Fanuc TP program (LS listing): DISTI_LINE_V1.LS

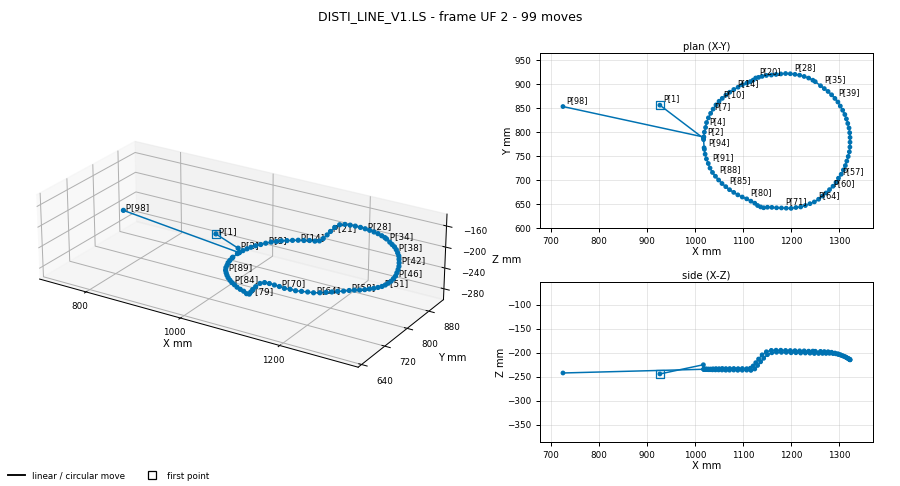
[picture p0: tool path of DISTI_LINE_V1.LS in frame UF 2, 99 of 99 moves have a stored position in this frame; points joined in program order, loops and branches not executed]
/PROG  DISTI_LINE_V1
/ATTR
OWNER		= MNEDITOR;
COMMENT		= "WeldPRO Auto-Gen";
PROG_SIZE	= 7109;
CREATE		= DATE 26-07-21  TIME 17:58:54;
MODIFIED	= DATE 26-07-21  TIME 18:14:06;
FILE_NAME	= DISTI_LI;
VERSION		= 0;
LINE_COUNT	= 113;
MEMORY_SIZE	= 7429;
PROTECT		= READ_WRITE;
TCD:  STACK_SIZE	= 0,
      TASK_PRIORITY	= 50,
      TIME_SLICE	= 0,
      BUSY_LAMP_OFF	= 0,
      ABORT_REQUEST	= 0,
      PAUSE_REQUEST	= 0;
DEFAULT_GROUP	= 1,*,*,*,*;
CONTROL_CODE	= 00000000 00000000;
/APPL
/MN
   1:  !WeldPRO Auto-Generated TPP ;
   2:  !Tor XL_176 _2, Feature1 ;
   3:   ;
   4:  UFRAME_NUM=2 ;
   5:  UTOOL_NUM=2 ;
   6:L P[1] 100mm/sec FINE    ;
   7:   ;
   8:  !Segment1 ;
   9:L P[2] 100mm/sec FINE    ;
  10:  CALL LASER_OFF    ;
  11:   ;
  12:L P[99] R[23:moving]mm/sec CNT100    ;
  13:   ;
  14:L P[3] R[23:moving]mm/sec CNT100    ;
  15:L P[4] R[23:moving]mm/sec CNT100    ;
  16:L P[5] R[23:moving]mm/sec CNT100    ;
  17:L P[6] R[23:moving]mm/sec CNT100    ;
  18:L P[7] R[23:moving]mm/sec CNT100    ;
  19:L P[8] R[23:moving]mm/sec CNT100    ;
  20:L P[9] R[23:moving]mm/sec CNT100    ;
  21:L P[10] R[23:moving]mm/sec CNT100    ;
  22:L P[11] R[23:moving]mm/sec CNT100    ;
  23:L P[12] R[23:moving]mm/sec CNT100    ;
  24:L P[13] R[23:moving]mm/sec CNT100    ;
  25:L P[14] R[23:moving]mm/sec CNT100    ;
  26:L P[15] R[23:moving]mm/sec CNT100    ;
  27:L P[16] R[23:moving]mm/sec CNT100    ;
  28:L P[17] R[23:moving]mm/sec CNT100    ;
  29:L P[18] R[23:moving]mm/sec CNT100    ;
  30:L P[19] R[23:moving]mm/sec CNT100    ;
  31:L P[20] R[23:moving]mm/sec CNT100    ;
  32:L P[21] R[23:moving]mm/sec CNT100    ;
  33:L P[22] R[23:moving]mm/sec CNT100    ;
  34:L P[23] R[23:moving]mm/sec CNT100    ;
  35:L P[24] R[23:moving]mm/sec CNT100    ;
  36:L P[25] R[23:moving]mm/sec CNT100    ;
  37:L P[26] R[23:moving]mm/sec CNT100    ;
  38:L P[27] R[23:moving]mm/sec CNT100    ;
  39:L P[28] R[23:moving]mm/sec CNT100    ;
  40:L P[29] R[23:moving]mm/sec CNT100    ;
  41:L P[30] R[23:moving]mm/sec CNT100    ;
  42:L P[31] R[23:moving]mm/sec CNT100    ;
  43:L P[32] R[23:moving]mm/sec CNT100    ;
  44:L P[33] R[23:moving]mm/sec CNT100    ;
  45:L P[34] R[23:moving]mm/sec CNT100    ;
  46:L P[35] R[23:moving]mm/sec CNT100    ;
  47:L P[36] R[23:moving]mm/sec CNT100    ;
  48:L P[37] R[23:moving]mm/sec CNT100    ;
  49:L P[38] R[23:moving]mm/sec CNT100    ;
  50:L P[39] R[23:moving]mm/sec CNT100    ;
  51:L P[40] R[23:moving]mm/sec CNT100    ;
  52:L P[41] R[23:moving]mm/sec CNT100    ;
  53:L P[42] R[23:moving]mm/sec CNT100    ;
  54:L P[43] R[23:moving]mm/sec CNT100    ;
  55:L P[44] R[23:moving]mm/sec CNT100    ;
  56:L P[45] R[23:moving]mm/sec CNT100    ;
  57:L P[46] R[23:moving]mm/sec CNT100    ;
  58:L P[47] R[23:moving]mm/sec CNT100    ;
  59:L P[48] R[23:moving]mm/sec CNT100    ;
  60:L P[49] R[23:moving]mm/sec CNT100    ;
  61:L P[50] R[23:moving]mm/sec CNT100    ;
  62:L P[51] R[23:moving]mm/sec CNT100    ;
  63:L P[52] R[23:moving]mm/sec CNT100    ;
  64:L P[53] R[23:moving]mm/sec CNT100    ;
  65:L P[54] R[23:moving]mm/sec CNT100    ;
  66:L P[55] R[23:moving]mm/sec CNT100    ;
  67:L P[56] R[23:moving]mm/sec CNT100    ;
  68:L P[57] R[23:moving]mm/sec CNT100    ;
  69:L P[58] R[23:moving]mm/sec CNT100    ;
  70:L P[59] R[23:moving]mm/sec CNT100    ;
  71:L P[60] R[23:moving]mm/sec CNT100    ;
  72:L P[61] R[23:moving]mm/sec CNT100    ;
  73:L P[62] R[23:moving]mm/sec CNT100    ;
  74:L P[63] R[23:moving]mm/sec CNT100    ;
  75:L P[64] R[23:moving]mm/sec CNT100    ;
  76:L P[65] R[23:moving]mm/sec CNT100    ;
  77:L P[66] R[23:moving]mm/sec CNT100    ;
  78:L P[67] R[23:moving]mm/sec CNT100    ;
  79:L P[68] R[23:moving]mm/sec CNT100    ;
  80:L P[69] R[23:moving]mm/sec CNT100    ;
  81:L P[70] R[23:moving]mm/sec CNT100    ;
  82:L P[71] R[23:moving]mm/sec CNT100    ;
  83:L P[72] R[23:moving]mm/sec CNT100    ;
  84:L P[73] R[23:moving]mm/sec CNT100    ;
  85:L P[74] R[23:moving]mm/sec CNT100    ;
  86:L P[75] R[23:moving]mm/sec CNT100    ;
  87:L P[76] R[23:moving]mm/sec CNT100    ;
  88:L P[77] R[23:moving]mm/sec CNT100    ;
  89:L P[78] R[23:moving]mm/sec CNT100    ;
  90:L P[79] R[23:moving]mm/sec CNT100    ;
  91:L P[80] R[23:moving]mm/sec CNT100    ;
  92:L P[81] R[23:moving]mm/sec CNT100    ;
  93:L P[82] R[23:moving]mm/sec CNT100    ;
  94:L P[83] R[23:moving]mm/sec CNT100    ;
  95:L P[84] R[23:moving]mm/sec CNT100    ;
  96:L P[85] R[23:moving]mm/sec CNT100    ;
  97:L P[86] R[23:moving]mm/sec CNT100    ;
  98:L P[87] R[23:moving]mm/sec CNT100    ;
  99:L P[88] R[23:moving]mm/sec CNT100    ;
 100:L P[89] R[23:moving]mm/sec CNT100    ;
 101:L P[90] R[23:moving]mm/sec CNT100    ;
 102:L P[91] R[23:moving]mm/sec CNT100    ;
 103:L P[92] R[23:moving]mm/sec CNT100    ;
 104:L P[93] R[23:moving]mm/sec CNT100    ;
 105:L P[94] R[23:moving]mm/sec CNT100    ;
 106:L P[95] R[23:moving]mm/sec CNT100    ;
 107:L P[96] R[23:moving]mm/sec CNT100    ;
 108:L P[97] R[23:moving]mm/sec FINE    ;
 109:  CALL LASER_OFF    ;
 110:   ;
 111:  !Feature Retreat ;
 112:L P[98] 100mm/sec FINE    ;
 113:  CALL ROTATE    ;
/POS
P[1]{
   GP1:
	UF : 2, UT : 2,		CONFIG : 'F D T, 0, 0, 0',
	X =   927.346  mm,	Y =   856.354  mm,	Z =  -244.034  mm,
	W =  -106.482 deg,	P =   -15.198 deg,	R =    86.345 deg
};
P[2]{
   GP1:
	UF : 2, UT : 2,		CONFIG : 'F D T, 0, 0, 0',
	X =  1017.849  mm,	Y =   787.602  mm,	Z =  -224.873  mm,
	W =  -106.491 deg,	P =   -15.193 deg,	R =    86.327 deg
};
P[3]{
   GP1:
	UF : 2, UT : 2,		CONFIG : 'F D T, 0, 0, 0',
	X =  1019.935  mm,	Y =   800.294  mm,	Z =  -233.990  mm,
	W =  -106.460 deg,	P =   -15.318 deg,	R =    81.648 deg
};
P[4]{
   GP1:
	UF : 2, UT : 2,		CONFIG : 'F D T, 0, 0, 0',
	X =  1022.444  mm,	Y =   809.956  mm,	Z =  -233.523  mm,
	W =  -106.425 deg,	P =   -15.445 deg,	R =    76.281 deg
};
P[5]{
   GP1:
	UF : 2, UT : 2,		CONFIG : 'F D T, 0, 0, 0',
	X =  1024.421  mm,	Y =   820.142  mm,	Z =  -233.847  mm,
	W =  -106.381 deg,	P =   -15.559 deg,	R =    71.464 deg
};
P[6]{
   GP1:
	UF : 2, UT : 2,		CONFIG : 'F D T, 0, 0, 0',
	X =  1028.297  mm,	Y =   829.982  mm,	Z =  -233.703  mm,
	W =  -106.310 deg,	P =   -15.698 deg,	R =    65.272 deg
};
P[7]{
   GP1:
	UF : 2, UT : 2,		CONFIG : 'F D T, 0, 0, 0',
	X =  1032.934  mm,	Y =   839.356  mm,	Z =  -233.745  mm,
	W =  -106.251 deg,	P =   -15.795 deg,	R =    60.811 deg
};
P[8]{
   GP1:
	UF : 2, UT : 2,		CONFIG : 'F D T, 0, 0, 0',
	X =  1038.061  mm,	Y =   848.132  mm,	Z =  -233.295  mm,
	W =  -106.174 deg,	P =   -15.897 deg,	R =    55.794 deg
};
P[9]{
   GP1:
	UF : 2, UT : 2,		CONFIG : 'F D T, 0, 0, 0',
	X =  1044.053  mm,	Y =   856.873  mm,	Z =  -232.984  mm,
	W =  -106.090 deg,	P =   -15.988 deg,	R =    50.970 deg
};
P[10]{
   GP1:
	UF : 2, UT : 2,		CONFIG : 'F D T, 0, 0, 0',
	X =  1050.502  mm,	Y =   864.509  mm,	Z =  -233.095  mm,
	W =  -106.027 deg,	P =   -16.056 deg,	R =    47.314 deg
};
P[11]{
   GP1:
	UF : 2, UT : 2,		CONFIG : 'F D T, 0, 0, 0',
	X =  1057.143  mm,	Y =   870.540  mm,	Z =  -232.650  mm,
	W =  -105.939 deg,	P =   -16.126 deg,	R =    42.935 deg
};
P[12]{
   GP1:
	UF : 2, UT : 2,		CONFIG : 'F D T, 0, 0, 0',
	X =  1064.674  mm,	Y =   877.253  mm,	Z =  -232.934  mm,
	W =  -105.872 deg,	P =   -16.175 deg,	R =    39.733 deg
};
P[13]{
   GP1:
	UF : 2, UT : 2,		CONFIG : 'F D T, 0, 0, 0',
	X =  1072.654  mm,	Y =   883.324  mm,	Z =  -232.851  mm,
	W =  -105.783 deg,	P =   -16.243 deg,	R =    35.484 deg
};
P[14]{
   GP1:
	UF : 2, UT : 2,		CONFIG : 'F D T, 0, 0, 0',
	X =  1081.152  mm,	Y =   888.974  mm,	Z =  -232.722  mm,
	W =  -105.683 deg,	P =   -16.290 deg,	R =    31.072 deg
};
P[15]{
   GP1:
	UF : 2, UT : 2,		CONFIG : 'F D T, 0, 0, 0',
	X =  1090.115  mm,	Y =   893.784  mm,	Z =  -232.991  mm,
	W =  -105.584 deg,	P =   -16.329 deg,	R =    26.914 deg
};
P[16]{
   GP1:
	UF : 2, UT : 2,		CONFIG : 'F D T, 0, 0, 0',
	X =  1098.940  mm,	Y =   898.687  mm,	Z =  -232.748  mm,
	W =  -105.545 deg,	P =   -16.341 deg,	R =    25.103 deg
};
P[17]{
   GP1:
	UF : 2, UT : 2,		CONFIG : 'F D T, 0, 0, 0',
	X =  1107.970  mm,	Y =   902.159  mm,	Z =  -233.094  mm,
	W =  -115.468 deg,	P =   -16.090 deg,	R =    30.046 deg
};
P[18]{
   GP1:
	UF : 2, UT : 2,		CONFIG : 'F D T, 0, 0, 0',
	X =  1115.546  mm,	Y =   905.308  mm,	Z =  -232.090  mm,
	W =  -126.721 deg,	P =   -15.366 deg,	R =    26.538 deg
};
P[19]{
   GP1:
	UF : 2, UT : 2,		CONFIG : 'F D T, 0, 0, 0',
	X =  1121.367  mm,	Y =   908.505  mm,	Z =  -227.368  mm,
	W =  -119.393 deg,	P =   -15.981 deg,	R =    16.221 deg
};
P[20]{
   GP1:
	UF : 2, UT : 2,		CONFIG : 'F D T, 0, 0, 0',
	X =  1126.751  mm,	Y =   912.917  mm,	Z =  -220.637  mm,
	W =  -115.329 deg,	P =   -16.208 deg,	R =    11.788 deg
};
P[21]{
   GP1:
	UF : 2, UT : 2,		CONFIG : 'F D T, 0, 0, 0',
	X =  1132.715  mm,	Y =   914.254  mm,	Z =  -213.028  mm,
	W =  -112.690 deg,	P =   -16.313 deg,	R =     9.687 deg
};
P[22]{
   GP1:
	UF : 2, UT : 2,		CONFIG : 'F D T, 0, 0, 0',
	X =  1140.073  mm,	Y =   916.305  mm,	Z =  -204.283  mm,
	W =  -110.089 deg,	P =   -16.384 deg,	R =     9.676 deg
};
P[23]{
   GP1:
	UF : 2, UT : 2,		CONFIG : 'F D T, 0, 0, 0',
	X =  1148.969  mm,	Y =   918.238  mm,	Z =  -197.811  mm,
	W =  -107.448 deg,	P =   -16.428 deg,	R =     8.430 deg
};
P[24]{
   GP1:
	UF : 2, UT : 2,		CONFIG : 'F D T, 0, 0, 0',
	X =  1159.237  mm,	Y =   919.017  mm,	Z =  -194.999  mm,
	W =  -105.451 deg,	P =   -16.442 deg,	R =     6.850 deg
};
P[25]{
   GP1:
	UF : 2, UT : 2,		CONFIG : 'F D T, 0, 0, 0',
	X =  1169.084  mm,	Y =   920.317  mm,	Z =  -194.637  mm,
	W =  -104.865 deg,	P =   -16.444 deg,	R =     5.674 deg
};
P[26]{
   GP1:
	UF : 2, UT : 2,		CONFIG : 'F D T, 0, 0, 0',
	X =  1178.939  mm,	Y =   921.340  mm,	Z =  -194.644  mm,
	W =  -104.885 deg,	P =   -16.444 deg,	R =     3.732 deg
};
P[27]{
   GP1:
	UF : 2, UT : 2,		CONFIG : 'F D T, 0, 0, 0',
	X =  1188.875  mm,	Y =   922.217  mm,	Z =  -195.137  mm,
	W =  -104.928 deg,	P =   -16.440 deg,	R =     -.482 deg
};
P[28]{
   GP1:
	UF : 2, UT : 2,		CONFIG : 'F D T, 0, 0, 0',
	X =  1198.726  mm,	Y =   921.678  mm,	Z =  -195.333  mm,
	W =  -104.977 deg,	P =   -16.425 deg,	R =    -5.295 deg
};
P[29]{
   GP1:
	UF : 2, UT : 2,		CONFIG : 'F D T, 0, 0, 0',
	X =  1208.426  mm,	Y =   920.468  mm,	Z =  -195.571  mm,
	W =  -105.026 deg,	P =   -16.401 deg,	R =   -10.039 deg
};
P[30]{
   GP1:
	UF : 2, UT : 2,		CONFIG : 'F D T, 0, 0, 0',
	X =  1218.075  mm,	Y =   918.762  mm,	Z =  -195.921  mm,
	W =  -105.069 deg,	P =   -16.371 deg,	R =   -14.284 deg
};
P[31]{
   GP1:
	UF : 2, UT : 2,		CONFIG : 'F D T, 0, 0, 0',
	X =  1227.533  mm,	Y =   916.082  mm,	Z =  -195.973  mm,
	W =  -105.112 deg,	P =   -16.334 deg,	R =   -18.515 deg
};
P[32]{
   GP1:
	UF : 2, UT : 2,		CONFIG : 'F D T, 0, 0, 0',
	X =  1236.897  mm,	Y =   912.747  mm,	Z =  -196.590  mm,
	W =  -105.156 deg,	P =   -16.287 deg,	R =   -22.931 deg
};
P[33]{
   GP1:
	UF : 2, UT : 2,		CONFIG : 'F D T, 0, 0, 0',
	X =  1245.612  mm,	Y =   908.325  mm,	Z =  -196.471  mm,
	W =  -105.219 deg,	P =   -16.204 deg,	R =   -29.417 deg
};
P[34]{
   GP1:
	UF : 2, UT : 2,		CONFIG : 'F D T, 0, 0, 0',
	X =  1250.569  mm,	Y =   905.277  mm,	Z =  -196.787  mm,
	W =  -105.326 deg,	P =   -16.106 deg,	R =   -35.234 deg
};
P[35]{
   GP1:
	UF : 2, UT : 2,		CONFIG : 'F D T, 0, 0, 0',
	X =  1261.597  mm,	Y =   896.794  mm,	Z =  -197.084  mm,
	W =  -105.307 deg,	P =   -16.055 deg,	R =   -38.974 deg
};
P[36]{
   GP1:
	UF : 2, UT : 2,		CONFIG : 'F D T, 0, 0, 0',
	X =  1269.439  mm,	Y =   890.850  mm,	Z =  -197.514  mm,
	W =  -105.304 deg,	P =   -16.061 deg,	R =   -38.624 deg
};
P[37]{
   GP1:
	UF : 2, UT : 2,		CONFIG : 'F D T, 0, 0, 0',
	X =  1277.298  mm,	Y =   884.903  mm,	Z =  -197.829  mm,
	W =  -105.460 deg,	P =   -15.949 deg,	R =   -44.737 deg
};
P[38]{
   GP1:
	UF : 2, UT : 2,		CONFIG : 'F D T, 0, 0, 0',
	X =  1284.611  mm,	Y =   877.969  mm,	Z =  -198.885  mm,
	W =  -105.652 deg,	P =   -15.892 deg,	R =   -47.603 deg
};
P[39]{
   GP1:
	UF : 2, UT : 2,		CONFIG : 'F D T, 0, 0, 0',
	X =  1291.497  mm,	Y =   870.412  mm,	Z =  -200.508  mm,
	W =  -106.194 deg,	P =   -15.794 deg,	R =   -52.149 deg
};
P[40]{
   GP1:
	UF : 2, UT : 2,		CONFIG : 'F D T, 0, 0, 0',
	X =  1297.727  mm,	Y =   862.952  mm,	Z =  -201.956  mm,
	W =  -106.906 deg,	P =   -15.690 deg,	R =   -56.548 deg
};
P[41]{
   GP1:
	UF : 2, UT : 2,		CONFIG : 'F D T, 0, 0, 0',
	X =  1302.749  mm,	Y =   854.499  mm,	Z =  -203.792  mm,
	W =  -107.559 deg,	P =   -15.603 deg,	R =   -60.015 deg
};
P[42]{
   GP1:
	UF : 2, UT : 2,		CONFIG : 'F D T, 0, 0, 0',
	X =  1307.690  mm,	Y =   845.800  mm,	Z =  -206.094  mm,
	W =  -108.250 deg,	P =   -15.507 deg,	R =   -63.574 deg
};
P[43]{
   GP1:
	UF : 2, UT : 2,		CONFIG : 'F D T, 0, 0, 0',
	X =  1312.181  mm,	Y =   836.891  mm,	Z =  -208.095  mm,
	W =  -109.123 deg,	P =   -15.380 deg,	R =   -68.091 deg
};
P[44]{
   GP1:
	UF : 2, UT : 2,		CONFIG : 'F D T, 0, 0, 0',
	X =  1315.462  mm,	Y =   827.755  mm,	Z =  -209.918  mm,
	W =  -109.894 deg,	P =   -15.253 deg,	R =   -72.476 deg
};
P[45]{
   GP1:
	UF : 2, UT : 2,		CONFIG : 'F D T, 0, 0, 0',
	X =  1318.258  mm,	Y =   818.316  mm,	Z =  -211.674  mm,
	W =  -110.258 deg,	P =   -15.184 deg,	R =   -74.873 deg
};
P[46]{
   GP1:
	UF : 2, UT : 2,		CONFIG : 'F D T, 0, 0, 0',
	X =  1320.915  mm,	Y =   808.858  mm,	Z =  -213.290  mm,
	W =  -110.625 deg,	P =   -15.097 deg,	R =   -77.924 deg
};
P[47]{
   GP1:
	UF : 2, UT : 2,		CONFIG : 'F D T, 0, 0, 0',
	X =  1322.253  mm,	Y =   798.998  mm,	Z =  -213.962  mm,
	W =  -111.046 deg,	P =   -14.958 deg,	R =   -82.908 deg
};
P[48]{
   GP1:
	UF : 2, UT : 2,		CONFIG : 'F D T, 0, 0, 0',
	X =  1322.992  mm,	Y =   789.184  mm,	Z =  -214.656  mm,
	W =  -111.160 deg,	P =   -14.266 deg,	R =   -88.178 deg
};
P[49]{
   GP1:
	UF : 2, UT : 2,		CONFIG : 'F D T, 0, 0, 0',
	X =  1322.949  mm,	Y =   779.288  mm,	Z =  -214.535  mm,
	W =  -111.104 deg,	P =   -14.627 deg,	R =   -91.603 deg
};
P[50]{
   GP1:
	UF : 2, UT : 2,		CONFIG : 'F D T, 0, 0, 0',
	X =  1322.694  mm,	Y =   769.200  mm,	Z =  -213.952  mm,
	W =  -110.785 deg,	P =   -15.101 deg,	R =   -96.403 deg
};
P[51]{
   GP1:
	UF : 2, UT : 2,		CONFIG : 'F D T, 0, 0, 0',
	X =  1321.587  mm,	Y =   759.251  mm,	Z =  -213.085  mm,
	W =  -110.276 deg,	P =   -14.535 deg,	R =  -100.836 deg
};
P[52]{
   GP1:
	UF : 2, UT : 2,		CONFIG : 'F D T, 0, 0, 0',
	X =  1319.179  mm,	Y =   749.552  mm,	Z =  -211.671  mm,
	W =  -109.635 deg,	P =   -14.447 deg,	R =  -105.265 deg
};
P[53]{
   GP1:
	UF : 2, UT : 2,		CONFIG : 'F D T, 0, 0, 0',
	X =  1316.280  mm,	Y =   740.038  mm,	Z =  -210.276  mm,
	W =  -109.103 deg,	P =   -14.384 deg,	R =  -108.504 deg
};
P[54]{
   GP1:
	UF : 2, UT : 2,		CONFIG : 'F D T, 0, 0, 0',
	X =  1313.256  mm,	Y =   730.645  mm,	Z =  -208.544  mm,
	W =  -108.392 deg,	P =   -14.307 deg,	R =  -112.625 deg
};
P[55]{
   GP1:
	UF : 2, UT : 2,		CONFIG : 'F D T, 0, 0, 0',
	X =  1309.176  mm,	Y =   721.525  mm,	Z =  -207.037  mm,
	W =  -107.773 deg,	P =   -14.241 deg,	R =  -116.139 deg
};
P[56]{
   GP1:
	UF : 2, UT : 2,		CONFIG : 'F D T, 0, 0, 0',
	X =  1304.568  mm,	Y =   712.572  mm,	Z =  -205.463  mm,
	W =  -106.932 deg,	P =   -14.149 deg,	R =  -121.162 deg
};
P[57]{
   GP1:
	UF : 2, UT : 2,		CONFIG : 'F D T, 0, 0, 0',
	X =  1298.935  mm,	Y =   704.431  mm,	Z =  -203.750  mm,
	W =  -106.269 deg,	P =   -14.066 deg,	R =  -125.698 deg
};
P[58]{
   GP1:
	UF : 2, UT : 2,		CONFIG : 'F D T, 0, 0, 0',
	X =  1293.796  mm,	Y =   695.674  mm,	Z =  -202.230  mm,
	W =  -105.781 deg,	P =   -13.988 deg,	R =  -130.143 deg
};
P[59]{
   GP1:
	UF : 2, UT : 2,		CONFIG : 'F D T, 0, 0, 0',
	X =  1287.602  mm,	Y =   687.685  mm,	Z =  -201.692  mm,
	W =  -105.502 deg,	P =   -13.914 deg,	R =  -134.519 deg
};
P[60]{
   GP1:
	UF : 2, UT : 2,		CONFIG : 'F D T, 0, 0, 0',
	X =  1280.303  mm,	Y =   680.629  mm,	Z =  -201.139  mm,
	W =  -105.438 deg,	P =   -13.851 deg,	R =  -138.498 deg
};
P[61]{
   GP1:
	UF : 2, UT : 2,		CONFIG : 'F D T, 0, 0, 0',
	X =  1273.069  mm,	Y =   673.682  mm,	Z =  -201.344  mm,
	W =  -105.428 deg,	P =   -13.829 deg,	R =  -139.977 deg
};
P[62]{
   GP1:
	UF : 2, UT : 2,		CONFIG : 'F D T, 0, 0, 0',
	X =  1265.718  mm,	Y =   667.186  mm,	Z =  -201.284  mm,
	W =  -105.443 deg,	P =   -13.863 deg,	R =  -137.727 deg
};
P[63]{
   GP1:
	UF : 2, UT : 2,		CONFIG : 'F D T, 0, 0, 0',
	X =  1257.613  mm,	Y =   660.607  mm,	Z =  -201.395  mm,
	W =  -105.373 deg,	P =   -13.729 deg,	R =  -147.436 deg
};
P[64]{
   GP1:
	UF : 2, UT : 2,		CONFIG : 'F D T, 0, 0, 0',
	X =  1248.737  mm,	Y =   655.076  mm,	Z =  -201.447  mm,
	W =  -105.298 deg,	P =   -13.637 deg,	R =  -156.529 deg
};
P[65]{
   GP1:
	UF : 2, UT : 2,		CONFIG : 'F D T, 0, 0, 0',
	X =  1239.622  mm,	Y =   651.403  mm,	Z =  -200.843  mm,
	W =  -105.278 deg,	P =   -13.619 deg,	R =  -158.873 deg
};
P[66]{
   GP1:
	UF : 2, UT : 2,		CONFIG : 'F D T, 0, 0, 0',
	X =  1229.976  mm,	Y =   647.581  mm,	Z =  -200.522  mm,
	W =  -105.242 deg,	P =   -13.593 deg,	R =  -162.872 deg
};
P[67]{
   GP1:
	UF : 2, UT : 2,		CONFIG : 'F D T, 0, 0, 0',
	X =  1220.279  mm,	Y =   644.529  mm,	Z =  -200.573  mm,
	W =  -105.204 deg,	P =   -13.573 deg,	R =  -166.917 deg
};
P[68]{
   GP1:
	UF : 2, UT : 2,		CONFIG : 'F D T, 0, 0, 0',
	X =  1210.347  mm,	Y =   643.413  mm,	Z =  -199.912  mm,
	W =  -105.160 deg,	P =   -13.560 deg,	R =  -171.451 deg
};
P[69]{
   GP1:
	UF : 2, UT : 2,		CONFIG : 'F D T, 0, 0, 0',
	X =  1200.315  mm,	Y =   641.642  mm,	Z =  -200.013  mm,
	W =  -105.114 deg,	P =   -13.556 deg,	R =  -176.195 deg
};
P[70]{
   GP1:
	UF : 2, UT : 2,		CONFIG : 'F D T, 0, 0, 0',
	X =  1190.252  mm,	Y =   642.001  mm,	Z =  -199.228  mm,
	W =  -105.069 deg,	P =   -13.561 deg,	R =   179.311 deg
};
P[71]{
   GP1:
	UF : 2, UT : 2,		CONFIG : 'F D T, 0, 0, 0',
	X =  1180.270  mm,	Y =   642.513  mm,	Z =  -199.122  mm,
	W =  -105.038 deg,	P =   -13.569 deg,	R =   176.231 deg
};
P[72]{
   GP1:
	UF : 2, UT : 2,		CONFIG : 'F D T, 0, 0, 0',
	X =  1170.162  mm,	Y =   642.835  mm,	Z =  -199.050  mm,
	W =  -105.170 deg,	P =   -13.572 deg,	R =   175.317 deg
};
P[73]{
   GP1:
	UF : 2, UT : 2,		CONFIG : 'F D T, 0, 0, 0',
	X =  1160.299  mm,	Y =   643.728  mm,	Z =  -200.052  mm,
	W =  -106.961 deg,	P =   -13.569 deg,	R =   174.549 deg
};
P[74]{
   GP1:
	UF : 2, UT : 2,		CONFIG : 'F D T, 0, 0, 0',
	X =  1151.164  mm,	Y =   643.988  mm,	Z =  -203.993  mm,
	W =  -109.346 deg,	P =   -13.539 deg,	R =   174.478 deg
};
P[75]{
   GP1:
	UF : 2, UT : 2,		CONFIG : 'F D T, 0, 0, 0',
	X =  1143.276  mm,	Y =   642.913  mm,	Z =  -211.490  mm,
	W =  -112.145 deg,	P =   -13.468 deg,	R =   175.272 deg
};
P[76]{
   GP1:
	UF : 2, UT : 2,		CONFIG : 'F D T, 0, 0, 0',
	X =  1136.911  mm,	Y =   644.638  mm,	Z =  -218.791  mm,
	W =  -114.824 deg,	P =   -13.371 deg,	R =   175.449 deg
};
P[77]{
   GP1:
	UF : 2, UT : 2,		CONFIG : 'F D T, 0, 0, 0',
	X =  1130.669  mm,	Y =   647.592  mm,	Z =  -226.370  mm,
	W =  -120.114 deg,	P =   -13.109 deg,	R =   172.293 deg
};
P[78]{
   GP1:
	UF : 2, UT : 2,		CONFIG : 'F D T, 0, 0, 0',
	X =  1124.765  mm,	Y =   652.366  mm,	Z =  -233.718  mm,
	W =  -126.491 deg,	P =   -12.649 deg,	R =   168.032 deg
};
P[79]{
   GP1:
	UF : 2, UT : 2,		CONFIG : 'F D T, 0, 0, 0',
	X =  1116.705  mm,	Y =   656.648  mm,	Z =  -236.623  mm,
	W =  -119.899 deg,	P =   -13.263 deg,	R =   157.916 deg
};
P[80]{
   GP1:
	UF : 2, UT : 2,		CONFIG : 'F D T, 0, 0, 0',
	X =  1107.995  mm,	Y =   661.424  mm,	Z =  -236.113  mm,
	W =  -106.920 deg,	P =   -13.744 deg,	R =   154.284 deg
};
P[81]{
   GP1:
	UF : 2, UT : 2,		CONFIG : 'F D T, 0, 0, 0',
	X =  1098.735  mm,	Y =   665.244  mm,	Z =  -236.345  mm,
	W =  -105.725 deg,	P =   -13.738 deg,	R =   155.031 deg
};
P[82]{
   GP1:
	UF : 2, UT : 2,		CONFIG : 'F D T, 0, 0, 0',
	X =  1089.463  mm,	Y =   669.765  mm,	Z =  -236.398  mm,
	W =  -105.804 deg,	P =   -13.784 deg,	R =   151.515 deg
};
P[83]{
   GP1:
	UF : 2, UT : 2,		CONFIG : 'F D T, 0, 0, 0',
	X =  1080.959  mm,	Y =   674.925  mm,	Z =  -235.970  mm,
	W =  -105.884 deg,	P =   -13.836 deg,	R =   147.827 deg
};
P[84]{
   GP1:
	UF : 2, UT : 2,		CONFIG : 'F D T, 0, 0, 0',
	X =  1072.242  mm,	Y =   680.510  mm,	Z =  -236.228  mm,
	W =  -105.989 deg,	P =   -13.919 deg,	R =   142.627 deg
};
P[85]{
   GP1:
	UF : 2, UT : 2,		CONFIG : 'F D T, 0, 0, 0',
	X =  1064.419  mm,	Y =   686.813  mm,	Z =  -236.257  mm,
	W =  -106.066 deg,	P =   -13.990 deg,	R =   138.574 deg
};
P[86]{
   GP1:
	UF : 2, UT : 2,		CONFIG : 'F D T, 0, 0, 0',
	X =  1056.599  mm,	Y =   693.321  mm,	Z =  -235.897  mm,
	W =  -106.118 deg,	P =   -14.044 deg,	R =   135.639 deg
};
P[87]{
   GP1:
	UF : 2, UT : 2,		CONFIG : 'F D T, 0, 0, 0',
	X =  1049.526  mm,	Y =   700.669  mm,	Z =  -235.706  mm,
	W =  -106.192 deg,	P =   -14.130 deg,	R =   131.212 deg
};
P[88]{
   GP1:
	UF : 2, UT : 2,		CONFIG : 'F D T, 0, 0, 0',
	X =  1042.957  mm,	Y =   708.418  mm,	Z =  -235.654  mm,
	W =  -106.261 deg,	P =   -14.227 deg,	R =   126.545 deg
};
P[89]{
   GP1:
	UF : 2, UT : 2,		CONFIG : 'F D T, 0, 0, 0',
	X =  1036.787  mm,	Y =   716.399  mm,	Z =  -235.538  mm,
	W =  -106.325 deg,	P =   -14.335 deg,	R =   121.649 deg
};
P[90]{
   GP1:
	UF : 2, UT : 2,		CONFIG : 'F D T, 0, 0, 0',
	X =  1031.667  mm,	Y =   725.439  mm,	Z =  -235.241  mm,
	W =  -106.396 deg,	P =   -14.486 deg,	R =   115.073 deg
};
P[91]{
   GP1:
	UF : 2, UT : 2,		CONFIG : 'F D T, 0, 0, 0',
	X =  1028.052  mm,	Y =   735.007  mm,	Z =  -235.230  mm,
	W =  -106.437 deg,	P =   -14.604 deg,	R =   110.157 deg
};
P[92]{
   GP1:
	UF : 2, UT : 2,		CONFIG : 'F D T, 0, 0, 0',
	X =  1024.184  mm,	Y =   744.481  mm,	Z =  -234.981  mm,
	W =  -106.467 deg,	P =   -14.723 deg,	R =   105.309 deg
};
P[93]{
   GP1:
	UF : 2, UT : 2,		CONFIG : 'F D T, 0, 1, 0',
	X =  1021.498  mm,	Y =   754.386  mm,	Z =  -235.076  mm,
	W =  -106.486 deg,	P =   -14.842 deg,	R =   100.517 deg
};
P[94]{
   GP1:
	UF : 2, UT : 2,		CONFIG : 'F D T, 0, 1, 0',
	X =  1019.941  mm,	Y =   764.417  mm,	Z =  -234.547  mm,
	W =  -106.495 deg,	P =   -14.962 deg,	R =    95.764 deg
};
P[95]{
   GP1:
	UF : 2, UT : 2,		CONFIG : 'F D T, 0, 1, 0',
	X =  1019.333  mm,	Y =   767.685  mm,	Z =  -234.367  mm,
	W =  -106.506 deg,	P =   -15.000 deg,	R =    94.231 deg
};
P[96]{
   GP1:
	UF : 2, UT : 2,		CONFIG : 'F D T, 0, 1, 0',
	X =  1018.300  mm,	Y =   784.661  mm,	Z =  -234.230  mm,
	W =  -106.482 deg,	P =   -15.197 deg,	R =    86.402 deg
};
P[97]{
   GP1:
	UF : 2, UT : 2,		CONFIG : 'F D T, 0, 1, 0',
	X =  1018.683  mm,	Y =   790.013  mm,	Z =  -234.290  mm,
	W =  -106.482 deg,	P =   -15.198 deg,	R =    86.345 deg
};
P[98]{
   GP1:
	UF : 2, UT : 2,		CONFIG : 'F D T, 0, 1, 0',
	X =   725.689  mm,	Y =   853.506  mm,	Z =  -242.034  mm,
	W =  -106.487 deg,	P =   -15.200 deg,	R =    86.348 deg
};
P[99]{
   GP1:
	UF : 2, UT : 2,		CONFIG : 'F D T, 0, 0, 0',
	X =  1018.712  mm,	Y =   790.192  mm,	Z =  -234.057  mm,
	W =  -106.495 deg,	P =   -15.194 deg,	R =    86.332 deg
};
/END
